PROGRAM PRG_LVCP2_Group6
VAR
    // Function Block Instance
    fbContactor: FB_ContactorControl;

    // Contactor 1 IO Structure  
    stContactor_IO: ST_ContactorIO;
    
    // Başlangıç konfigürasyonu için flag
    bContactorInitDone: BOOL := FALSE;
    bCapacitorInitDone: BOOL := FALSE;	
END_VAR



	M_Contactor();
	
	M_Capacitor();

METHOD M_Capacitor : BOOL
VAR
    nGroupIndex : INT;
END_VAR

nGroupIndex := 5;  // Grup 6 için index

IF NOT bCapacitorInitDone THEN
    // Grup 6 değerlerini ata
    GVL_LVCP2.astCompensationGroups[nGroupIndex].rPower := 25.0;
    GVL_LVCP2.astCompensationGroups[nGroupIndex].rVoltage := 450.0;
    GVL_LVCP2.astCompensationGroups[nGroupIndex].nQuantity := 3;
    GVL_LVCP2.astCompensationGroups[nGroupIndex].sTagPrefix := '+EP7-31C1';
    GVL_LVCP2.astCompensationGroups[nGroupIndex].sProductCode := 'ENT.CXD-450-25';
    
    bCapacitorInitDone := TRUE;
END_IF

// Grup 6 aktif durumu
GVL_LVCP2.abGroupActive[nGroupIndex] := stContactor_IO.bFeedback;

M_Capacitor := TRUE;
END_METHOD

METHOD M_Contactor : BOOL
VAR_INPUT
END_VAR
IF NOT bContactorInitDone THEN
    // Konfigürasyon parametreleri
    GVL_LVCP2.stGroup6_ContactorHMI.stConfig.sProjectCode := '+EP7-30K1';
    GVL_LVCP2.stGroup6_ContactorHMI.stConfig.sProductCode := 'ABB 1SFL547002R1311';
    GVL_LVCP2.stGroup6_ContactorHMI.stConfig.rRatedCurrent := 265.0;
    GVL_LVCP2.stGroup6_ContactorHMI.stConfig.rRatedVoltage := 1000.0;
    GVL_LVCP2.stGroup6_ContactorHMI.stConfig.nPhaseCount := 3;
    GVL_LVCP2.stGroup6_ContactorHMI.stConfig.tFeedbackDelay := T#500MS;
    GVL_LVCP2.stGroup6_ContactorHMI.stConfig.tWeldedDelay := T#2S;
    GVL_LVCP2.stGroup6_ContactorHMI.stConfig.dwOperationLimit := 100000;
    
    // Başlangıç bakım sayacı
    GVL_LVCP2.stGroup6_ContactorHMI.stStatistics.dwRemainingOperations := GVL_LVCP2.stGroup6_ContactorHMI.stConfig.dwOperationLimit;
    
    bContactorInitDone := TRUE;
END_IF

// Function Block Çağrısı
fbContactor(
    // Fiziksel Girişler
    bFeedback := stContactor_IO.bFeedback,
    bPLCControl := stContactor_IO.bPLCControl,
    
    // Güvenlik Girişleri
    bSafetyLoop := GVL_Alarm.bSafetyLoop,
    bInterlock := FALSE,
    
    // Sistem Girişleri
    bMasterReset := GVL_Alarm.bMasterReset,
    
    // HMI Bağlantısı
    stHMI := GVL_LVCP2.stGroup6_ContactorHMI,
    
    // Fiziksel Çıkış
    bOutput => stContactor_IO.bOutput
);

M_Contactor := TRUE;
END_METHOD

END_PROGRAM

(* stored: Version 1.1.0.1, ProductVersion 3.1.4024.14
   POU PRG_LVCP2_Group6: Id {35015fb6-54c8-4930-b0a3-13bfcd990270}, SpecialFunc None
   Method M_Capacitor: Id {f0fd80d6-8007-4fc4-9274-fe081bed93cc}
   Method M_Contactor: Id {09f83265-976e-4002-af17-bb9ca778091a} *)
